FUNCTION Rad2Deg : LREAL
VAR_INPUT
	rad: LREAL;
END_VAR
VAR
END_VAR

Rad2Deg := rad / PI * 180.0;

END_FUNCTION

(* stored: Version 1.1.0.1, ProductVersion 3.1.4024.12
   POU Rad2Deg: Id {a320a001-4311-4bc7-9be8-f3dc9b2d884e}, SpecialFunc None *)
